// TIA Portal V17 export
// export: Created 2024-06-14T09:52:15.1112925Z, ExportSetting WithDefaults, DisplayName Totally Integrated Automation Portal, DisplayVersion V17, DisplayName TIA Portal Openness, DisplayVersion V17, DisplayName TIA Portal Version Control Interface, DisplayVersion V17, DisplayName Simotion SCOUT TIA, DisplayVersion 5.4.3.0, DisplayName SINAMICS Startdrive Advanced, DisplayVersion V17 SP1 Update 1, DisplayName SINAMICS Startdrive G110M, G120, G120C, G120D, G120P, G115D, DisplayVersion V17 SP1 Update 1, DisplayName SINAMICS Startdrive G130, G150, S120, S150, SINAMICS MV, S210, DisplayVersion V17 SP1 Update 1, DisplayName STEP 7 Professional, DisplayVersion V17, DisplayName STEP 7 Safety, DisplayVersion V17, DisplayName WinCC Professional, DisplayVersion V17
ORGANIZATION_BLOCK "Main"   // OB1, LAD, ProgramCycle
TITLE = "Main Program Sweep (Cycle)"
{ S7_Optimized_Access := 'TRUE' }
VERSION : 0.1
// stored: AutoNumber true, IsIECCheckEnabled false, SetENOAutomatically false
   VAR_INPUT
      Initial_Call : Bool;   // Initial call of this OB
      Remanence : Bool;   // =True, if remanent data are available
   END_VAR
   VAR_TEMP
      temp : Int;
   END_VAR
   VAR_TEMP   // added for the SCL form of the ladder/FBD networks
      _w1 : Bool;
      _w2 : Bool;
      _w3 : Bool;
      _w4 : Bool;
   END_VAR
BEGIN

REGION Network 1
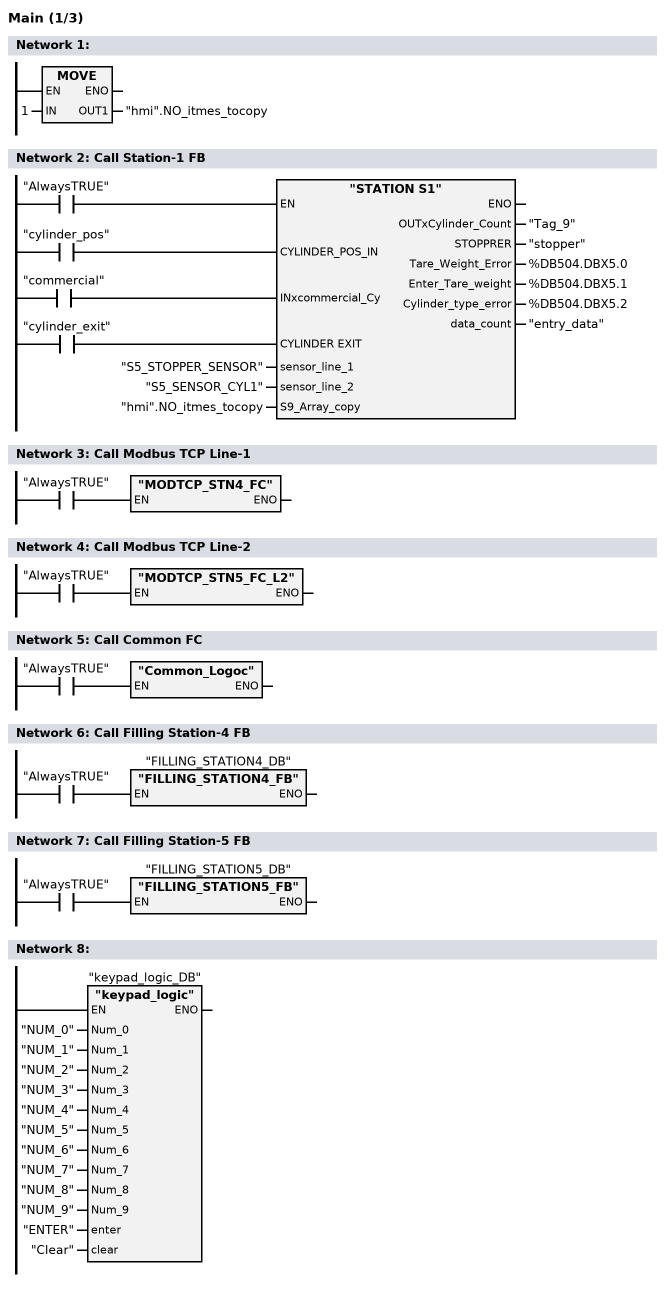
   RUNG wire#powerrail
      Move(in := 1, out1 => "hmi".NO_itmes_tocopy)
   END_RUNG
   // the same network as SCL:
   "hmi".NO_itmes_tocopy := 1;
END_REGION

REGION Network 2: Call Station-1 FB
   RUNG wire#powerrail
      Contact( "AlwaysTRUE" )
      "STATION S1"(CYLINDER_POS_IN := wire#w1, INxcommercial_Cy := wire#w2, "CYLINDER EXIT" := wire#w3, sensor_line_1 := "S5_STOPPER_SENSOR", sensor_line_2 := "S5_SENSOR_CYL1", S9_Array_copy := "hmi".NO_itmes_tocopy, OUTxCylinder_Count => "Tag_9", STOPPRER => "stopper", Tare_Weight_Error => %DB504.DBX5.0, Enter_Tare_weight => %DB504.DBX5.1, Cylinder_type_error => %DB504.DBX5.2, data_count => "entry_data")
   END_RUNG
   RUNG wire#powerrail
      Contact( "cylinder_pos" )
   END_RUNG wire#w1
   RUNG wire#powerrail
      Contact( "commercial" )
   END_RUNG wire#w2
   RUNG wire#powerrail
      Contact( "cylinder_exit" )
   END_RUNG wire#w3
   // the same network as SCL:
   IF "AlwaysTRUE" THEN
       "STATION S1"(CYLINDER_POS_IN := "cylinder_pos",
                    INxcommercial_Cy := "commercial",
                    "CYLINDER EXIT" := "cylinder_exit",
                    sensor_line_1 := "S5_STOPPER_SENSOR",
                    sensor_line_2 := "S5_SENSOR_CYL1",
                    S9_Array_copy := "hmi".NO_itmes_tocopy,
                    OUTxCylinder_Count => "Tag_9",
                    STOPPRER => "stopper",
                    Tare_Weight_Error => %DB504.DBX5.0,
                    Enter_Tare_weight => %DB504.DBX5.1,
                    Cylinder_type_error => %DB504.DBX5.2,
                    data_count => "entry_data");
   END_IF;
END_REGION

REGION Network 3: Call Modbus TCP Line-1
   RUNG wire#powerrail
      Contact( "AlwaysTRUE" )
      "MODTCP_STN4_FC"()
   END_RUNG
   // the same network as SCL:
   IF "AlwaysTRUE" THEN "MODTCP_STN4_FC"(); END_IF;
END_REGION

REGION Network 4: Call Modbus TCP Line-2
   RUNG wire#powerrail
      Contact( "AlwaysTRUE" )
      "MODTCP_STN5_FC_L2"()
   END_RUNG
   // the same network as SCL:
   IF "AlwaysTRUE" THEN "MODTCP_STN5_FC_L2"(); END_IF;
END_REGION

REGION Network 5: Call Common FC
   RUNG wire#powerrail
      Contact( "AlwaysTRUE" )
      "Common_Logoc"()
   END_RUNG
   // the same network as SCL:
   IF "AlwaysTRUE" THEN "Common_Logoc"(); END_IF;
END_REGION

REGION Network 6: Call Filling Station-4 FB
   RUNG wire#powerrail
      Contact( "AlwaysTRUE" )
      "FILLING_STATION4_DB"()
   END_RUNG
   // the same network as SCL:
   IF "AlwaysTRUE" THEN
       "FILLING_STATION4_DB"();   // "FILLING_STATION4_FB"
   END_IF;
END_REGION

REGION Network 7: Call Filling Station-5 FB
   RUNG wire#powerrail
      Contact( "AlwaysTRUE" )
      "FILLING_STATION5_DB"()
   END_RUNG
   // the same network as SCL:
   IF "AlwaysTRUE" THEN
       "FILLING_STATION5_DB"();   // "FILLING_STATION5_FB"
   END_IF;
END_REGION

REGION Network 8
   RUNG wire#powerrail
      "keypad_logic_DB"(Num_0 := "NUM_0", Num_1 := "NUM_1", Num_2 := "NUM_2", Num_3 := "NUM_3", Num_4 := "NUM_4", Num_5 := "NUM_5", Num_6 := "NUM_6", Num_7 := "NUM_7", Num_8 := "NUM_8", Num_9 := "NUM_9", enter := "ENTER", clear := "Clear")
   END_RUNG
   // the same network as SCL:
   "keypad_logic_DB"(Num_0 := "NUM_0",   // "keypad_logic"
                     Num_1 := "NUM_1",
                     Num_2 := "NUM_2",
                     Num_3 := "NUM_3",
                     Num_4 := "NUM_4",
                     Num_5 := "NUM_5",
                     Num_6 := "NUM_6",
                     Num_7 := "NUM_7",
                     Num_8 := "NUM_8",
                     Num_9 := "NUM_9",
                     enter := "ENTER",
                     clear := "Clear");
END_REGION

REGION Network 10: divde
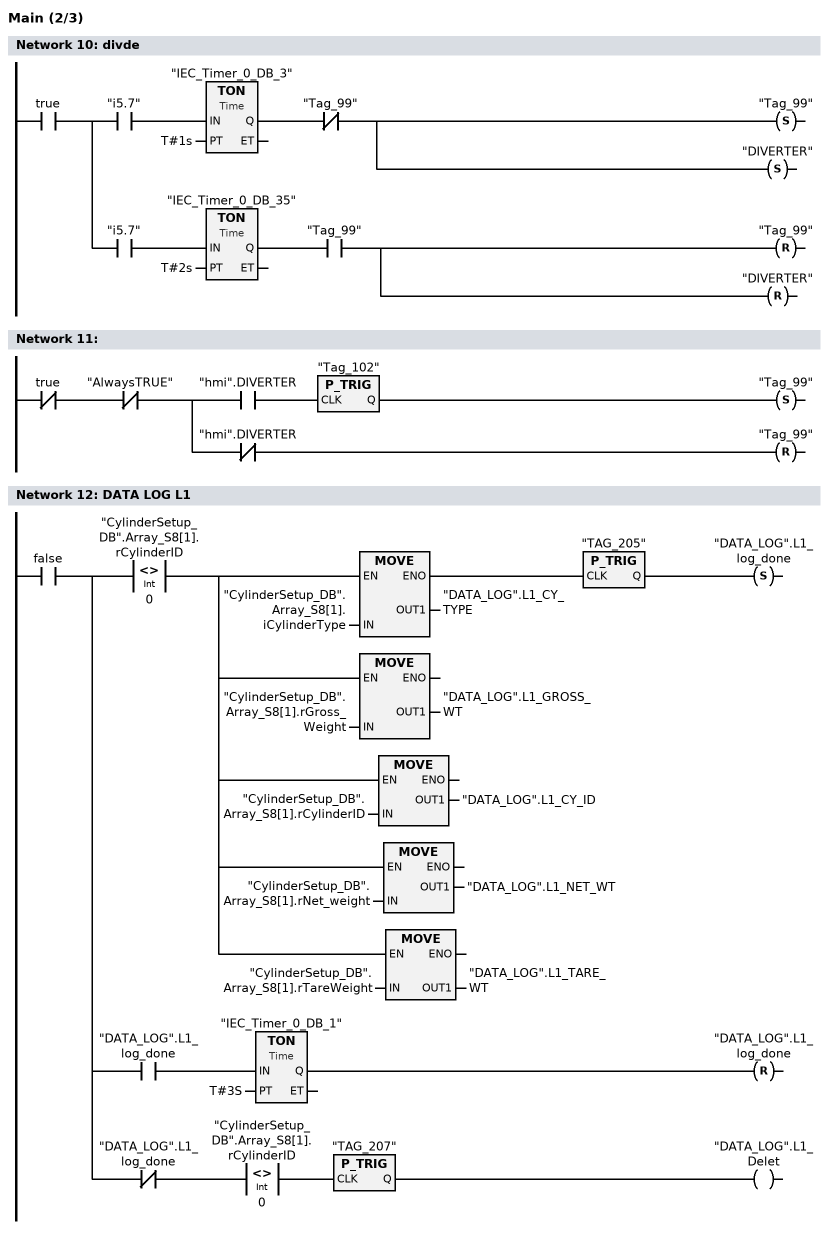
   RUNG wire#powerrail
      Contact( true )
      wire#w1
      Contact( "i5.7" )
      { S7_Templates := "time_type := Time" } "IEC_Timer_0_DB_3".TON(pt := T#1s, et =>)
      I_Contact( "Tag_99" )
      wire#w2
      S_Coil( "Tag_99" )
   END_RUNG
   RUNG wire#w2
      S_Coil( "DIVERTER" )
   END_RUNG
   RUNG wire#w1
      Contact( "i5.7" )
      { S7_Templates := "time_type := Time" } "IEC_Timer_0_DB_35".TON(pt := T#2s, et =>)
      Contact( "Tag_99" )
      wire#w3
      R_Coil( "Tag_99" )
   END_RUNG
   RUNG wire#w3
      R_Coil( "DIVERTER" )
   END_RUNG
   // the same network as SCL:
   "IEC_Timer_0_DB_3".TON(IN := true AND "i5.7", PT := T#1s);
   #_w1 := "IEC_Timer_0_DB_3".Q AND NOT "Tag_99";
   IF #_w1 THEN
       "Tag_99" := TRUE;
       "DIVERTER" := TRUE;
   END_IF;
   "IEC_Timer_0_DB_35".TON(IN := true AND "i5.7", PT := T#2s);
   #_w2 := "IEC_Timer_0_DB_35".Q AND "Tag_99";
   IF #_w2 THEN
       "Tag_99" := FALSE;
       "DIVERTER" := FALSE;
   END_IF;
END_REGION

REGION Network 11
   RUNG wire#powerrail
      I_Contact( true )
      I_Contact( "AlwaysTRUE" )
      wire#w1
      Contact( "hmi".DIVERTER )
      P_Trig( "Tag_102" )
      S_Coil( "Tag_99" )
   END_RUNG
   RUNG wire#w1
      I_Contact( "hmi".DIVERTER )
      R_Coil( "Tag_99" )
   END_RUNG
   // the same network as SCL:
   #_w1 := NOT true AND NOT "AlwaysTRUE";
   #_w2 := #_w1 AND "hmi".DIVERTER;
   #_w3 := #_w2 AND NOT "Tag_102";   // rising edge
   "Tag_102" := #_w2;
   IF #_w3 THEN "Tag_99" := TRUE; END_IF;
   IF #_w1 AND NOT "hmi".DIVERTER THEN "Tag_99" := FALSE; END_IF;
END_REGION

REGION Network 12: DATA LOG L1
   RUNG wire#powerrail
      Contact( false )
      wire#w1
      { S7_Templates := "SrcType := Int" } NE_Contact(in1 := "CylinderSetup_DB".Array_S8[1].rCylinderID, in2 := 0)
      wire#w2
      Move(in := "CylinderSetup_DB".Array_S8[1].iCylinderType, out1 => "DATA_LOG".L1_CY_TYPE)
      P_Trig( "TAG_205" )
      S_Coil( "DATA_LOG".L1_log_done )
   END_RUNG
   RUNG wire#w2
      Move(in := "CylinderSetup_DB".Array_S8[1].rGross_Weight, out1 => "DATA_LOG".L1_GROSS_WT)
   END_RUNG
   RUNG wire#w2
      Move(in := "CylinderSetup_DB".Array_S8[1].rCylinderID, out1 => "DATA_LOG".L1_CY_ID)
   END_RUNG
   RUNG wire#w2
      Move(in := "CylinderSetup_DB".Array_S8[1].rNet_weight, out1 => "DATA_LOG".L1_NET_WT)
   END_RUNG
   RUNG wire#w2
      Move(in := "CylinderSetup_DB".Array_S8[1].rTareWeight, out1 => "DATA_LOG".L1_TARE_WT)
   END_RUNG
   RUNG wire#w1
      Contact( "DATA_LOG".L1_log_done )
      { S7_Templates := "time_type := Time" } "IEC_Timer_0_DB_1".TON(pt := T#3S, et =>)
      R_Coil( "DATA_LOG".L1_log_done )
   END_RUNG
   RUNG wire#w1
      I_Contact( "DATA_LOG".L1_log_done )
      { S7_Templates := "SrcType := Int" } NE_Contact(in1 := "CylinderSetup_DB".Array_S8[1].rCylinderID, in2 := 0)
      P_Trig( "TAG_207" )
      Coil( "DATA_LOG".L1_Delet )
   END_RUNG
   // the same network as SCL:
   #_w1 := false AND ("CylinderSetup_DB".Array_S8[1].rCylinderID <> 0);
   IF #_w1 THEN "DATA_LOG".L1_CY_TYPE := "CylinderSetup_DB".Array_S8[1].iCylinderType; END_IF;
   #_w2 := #_w1 AND NOT "TAG_205";   // rising edge
   "TAG_205" := #_w1;
   IF #_w2 THEN "DATA_LOG".L1_log_done := TRUE; END_IF;
   IF #_w1 THEN
       "DATA_LOG".L1_GROSS_WT := "CylinderSetup_DB".Array_S8[1].rGross_Weight;
       "DATA_LOG".L1_CY_ID := "CylinderSetup_DB".Array_S8[1].rCylinderID;
       "DATA_LOG".L1_NET_WT := "CylinderSetup_DB".Array_S8[1].rNet_weight;
       "DATA_LOG".L1_TARE_WT := "CylinderSetup_DB".Array_S8[1].rTareWeight;
   END_IF;
   "IEC_Timer_0_DB_1".TON(IN := false AND "DATA_LOG".L1_log_done, PT := T#3S);
   IF "IEC_Timer_0_DB_1".Q THEN "DATA_LOG".L1_log_done := FALSE; END_IF;
   #_w3 := false AND NOT "DATA_LOG".L1_log_done AND ("CylinderSetup_DB".Array_S8[1].rCylinderID <> 0);
   #_w4 := #_w3 AND NOT "TAG_207";   // rising edge
   "TAG_207" := #_w3;
   "DATA_LOG".L1_Delet := #_w4;
END_REGION

REGION Network 13: DATA LOG L2
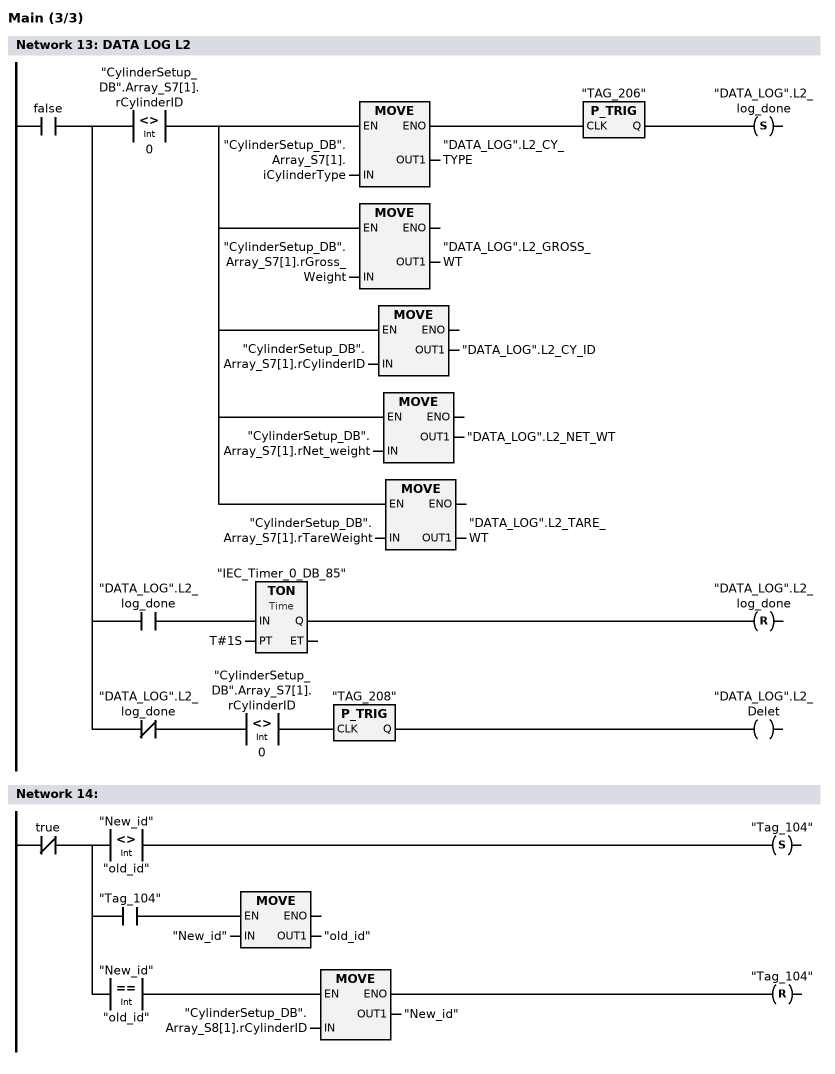
   RUNG wire#powerrail
      Contact( false )
      wire#w1
      { S7_Templates := "SrcType := Int" } NE_Contact(in1 := "CylinderSetup_DB".Array_S7[1].rCylinderID, in2 := 0)
      wire#w2
      Move(in := "CylinderSetup_DB".Array_S7[1].iCylinderType, out1 => "DATA_LOG".L2_CY_TYPE)
      P_Trig( "TAG_206" )
      S_Coil( "DATA_LOG".L2_log_done )
   END_RUNG
   RUNG wire#w2
      Move(in := "CylinderSetup_DB".Array_S7[1].rGross_Weight, out1 => "DATA_LOG".L2_GROSS_WT)
   END_RUNG
   RUNG wire#w2
      Move(in := "CylinderSetup_DB".Array_S7[1].rCylinderID, out1 => "DATA_LOG".L2_CY_ID)
   END_RUNG
   RUNG wire#w2
      Move(in := "CylinderSetup_DB".Array_S7[1].rNet_weight, out1 => "DATA_LOG".L2_NET_WT)
   END_RUNG
   RUNG wire#w2
      Move(in := "CylinderSetup_DB".Array_S7[1].rTareWeight, out1 => "DATA_LOG".L2_TARE_WT)
   END_RUNG
   RUNG wire#w1
      Contact( "DATA_LOG".L2_log_done )
      { S7_Templates := "time_type := Time" } "IEC_Timer_0_DB_85".TON(pt := T#1S, et =>)
      R_Coil( "DATA_LOG".L2_log_done )
   END_RUNG
   RUNG wire#w1
      I_Contact( "DATA_LOG".L2_log_done )
      { S7_Templates := "SrcType := Int" } NE_Contact(in1 := "CylinderSetup_DB".Array_S7[1].rCylinderID, in2 := 0)
      P_Trig( "TAG_208" )
      Coil( "DATA_LOG".L2_Delet )
   END_RUNG
   // the same network as SCL:
   #_w1 := false AND ("CylinderSetup_DB".Array_S7[1].rCylinderID <> 0);
   IF #_w1 THEN "DATA_LOG".L2_CY_TYPE := "CylinderSetup_DB".Array_S7[1].iCylinderType; END_IF;
   #_w2 := #_w1 AND NOT "TAG_206";   // rising edge
   "TAG_206" := #_w1;
   IF #_w2 THEN "DATA_LOG".L2_log_done := TRUE; END_IF;
   IF #_w1 THEN
       "DATA_LOG".L2_GROSS_WT := "CylinderSetup_DB".Array_S7[1].rGross_Weight;
       "DATA_LOG".L2_CY_ID := "CylinderSetup_DB".Array_S7[1].rCylinderID;
       "DATA_LOG".L2_NET_WT := "CylinderSetup_DB".Array_S7[1].rNet_weight;
       "DATA_LOG".L2_TARE_WT := "CylinderSetup_DB".Array_S7[1].rTareWeight;
   END_IF;
   "IEC_Timer_0_DB_85".TON(IN := false AND "DATA_LOG".L2_log_done, PT := T#1S);
   IF "IEC_Timer_0_DB_85".Q THEN "DATA_LOG".L2_log_done := FALSE; END_IF;
   #_w3 := false AND NOT "DATA_LOG".L2_log_done AND ("CylinderSetup_DB".Array_S7[1].rCylinderID <> 0);
   #_w4 := #_w3 AND NOT "TAG_208";   // rising edge
   "TAG_208" := #_w3;
   "DATA_LOG".L2_Delet := #_w4;
END_REGION

REGION Network 14
   RUNG wire#powerrail
      I_Contact( true )
      wire#w1
      { S7_Templates := "SrcType := Int" } NE_Contact(in1 := "New_id", in2 := "old_id")
      S_Coil( "Tag_104" )
   END_RUNG
   RUNG wire#w1
      Contact( "Tag_104" )
      Move(in := "New_id", out1 => "old_id")
   END_RUNG
   RUNG wire#w1
      { S7_Templates := "SrcType := Int" } EQ_Contact(in1 := "New_id", in2 := "old_id")
      Move(in := "CylinderSetup_DB".Array_S8[1].rCylinderID, out1 => "New_id")
      R_Coil( "Tag_104" )
   END_RUNG
   // the same network as SCL:
   IF NOT true AND ("New_id" <> "old_id") THEN "Tag_104" := TRUE; END_IF;
   IF NOT true AND "Tag_104" THEN "old_id" := "New_id"; END_IF;
   #_w1 := NOT true AND ("New_id" = "old_id");
   IF #_w1 THEN
       "New_id" := "CylinderSetup_DB".Array_S8[1].rCylinderID;
       "Tag_104" := FALSE;
   END_IF;
END_REGION
END_ORGANIZATION_BLOCK
